FUNCTION_BLOCK CL_AxisMCL1LeftBack EXTENDS CL_AxisMC
VAR
  objAxisDriver : CL_AxisDriverL1LeftBack;
END_VAR

SUPER^();

METHOD PUBLIC Init : BOOL
VAR_INPUT
  stIrrLine       : ST_LineReference;
  stAxisMotor_P	  : POINTER TO AXIS_REF;
  stAxisMaster_P  : POINTER TO AXIS_REF;
  stDriver        : POINTER TO ST_DriverAX8206_HWI;
END_VAR
Init := FALSE;
IF stDriver <> 0 THEN
  Init := objAxisDriver.Init(stDriver := stDriver);
  Init := Init AND SUPER^.InitMC(stIrrLine := stIrrLine, stAxisMotor_P := stAxisMotor_P, stAxisMaster_P := stAxisMaster_P, AxisDriver_P := ADR(objAxisDriver));
END_IF
END_METHOD

METHOD PROTECTED InitDefect : BOOL
InitDefect := SUPER^.InitDefect();
ADSLOGSTR(ADSLOG_MSGTYPE_LOG, 'CL_AxisMCL1LeftBack init defect','');
END_METHOD

METHOD PROTECTED InitParams : BOOL
VAR_INPUT
END_VAR
InitParams := SUPER^.InitParams();
_sWhichAxis := 'left(L1)-back';
_lrInverse := 1.0;
END_METHOD

END_FUNCTION_BLOCK

(* stored: Version 1.1.0.1, ProductVersion 3.1.4024.12
   POU CL_AxisMCL1LeftBack: Id {471b1620-a4eb-4e45-adf5-d1968ea43216}, SpecialFunc None
   Method Init: Id {3e9db96b-e5aa-4ca5-a506-118e65ab3d05}
   Method InitDefect: Id {eae795de-6055-4462-8fdf-b6c77b3c5095}
   Method InitParams: Id {fde22834-ed60-4fc7-bb5f-c3c336426d56} *)
